{attribute 'qualified_only'}
{attribute 'strict'}
TYPE E_WaitType :
(
    None      := 0,
    Time      := 1,
    Condition := 2
);
END_TYPE

(* stored: Version 1.1.0.1
   DUT E_WaitType: Id {4db9ff95-8ff6-4357-9c34-09b67956b168} *)
